ABB RobotStudio station: PaletizadoTPL2.rspag

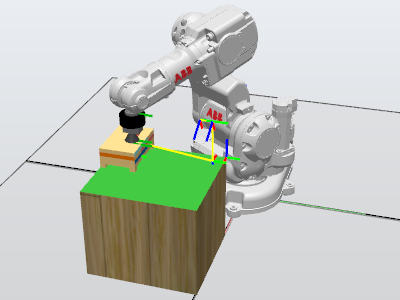
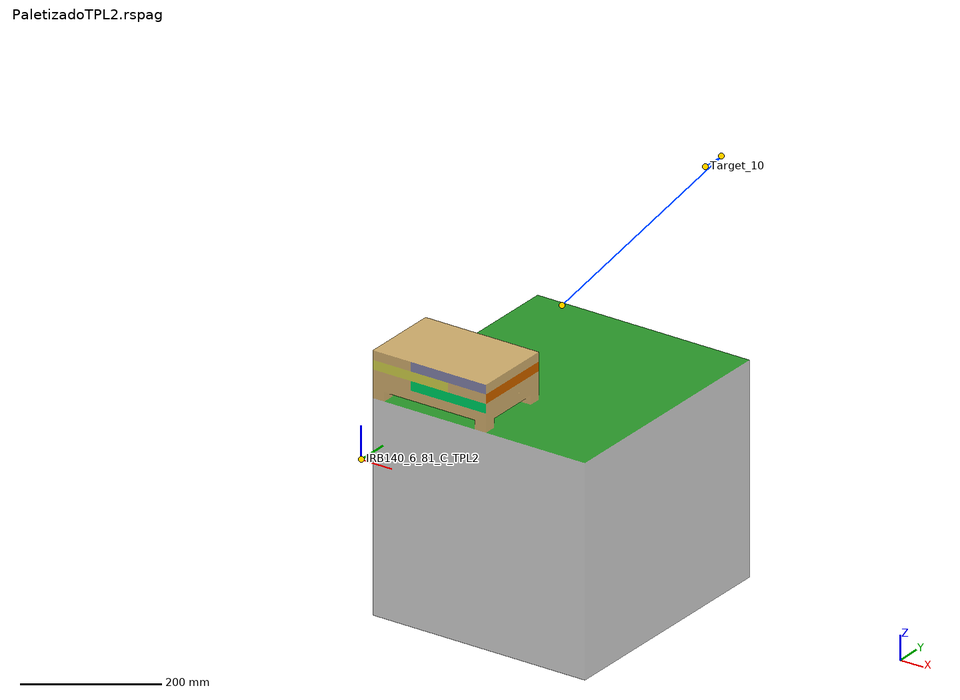
[picture v1: parts stored in the station drawn from their meshes, with robot base, taught points and paths (robot models come from the ABB library and are not in the file)]
--- station ---
Station Paletizado (saved by RobotStudio 25.5.11605.0)
Controller IRB140_6_81_TPL2
  mechanical unit ROB_1: IRB140_6_81_C_TPL2, 6 joints, base frame (0, 0, 0) mm
Layout (positions relative to the parent item):
  - Mesa [part], size 365 x 405 x 340 mm
  - Pallet [part], size 195 x 130 x 30 mm
  - Pieza1 [part] at (65, -275, 60) mm, size 130 x 65 x 15 mm
  - Pieza2 [part] at (795, -395, 45) mm, rotated rx 0 ry 0 rz -180 deg, size 130 x 65 x 15 mm
  - Pieza3 [part] at (305, -700, 30) mm, rotated rx 0 ry 0 rz 90 deg, size 130 x 65 x 15 mm
  - Pieza4 [part] at (730, -395, 0) mm, rotated rx 0 ry 0 rz -180 deg, size 130 x 65 x 15 mm
  - Pieza5 [part] at (0, -275, -15) mm, size 130 x 65 x 15 mm
  - Pieza6 [part] at (490, 30, -30) mm, rotated rx 0 ry 0 rz -90 deg, size 130 x 65 x 15 mm
  - Pieza7 [part] at (65, -275, -60) mm, size 130 x 65 x 15 mm
  - Pieza8 [part] at (795, -395, -75) mm, rotated rx 0 ry 0 rz -180 deg, size 130 x 65 x 15 mm
  - Pieza9 [part] at (305, -700, -90) mm, rotated rx 0 ry 0 rz 90 deg, size 130 x 65 x 15 mm
  - Sopapa [mechanism] at (430, -297.5, 533) mm, rotated rx -180 ry 0 rz 180 deg
      TCP Sopapa at (0, -5, 103) mm
      links: Sopapa
  - IRB140_6_81_C_TPL2 [mechanism, from %ABB.RobotStudio.Models.IRB140%\IRB140_6_81_C_G_03.rslib] at (0, 0, 0) mm; joint values [-0.6052, 0.2446, 0.0306, 0, 1.2955, -0.6052] (rad or m)
Attachment: Sopapa is attached to IRB140_6_81_C_TPL2 / Link6
Attachment: EsquinaPalet is attached to Pallet
EventTableEntry 1212: Group=, Trigger=DO_Sopapa 1213, Actions=[EventTableActionAttach 1214], Comment=, ActivationMode=2, Cyclic=false
EventTableTriggerIO 1213: IOValue=[1], IRC5Controller=? -1, Operator=0, SignalSource=IRB140_6_81_TPL2 1258
EventTableActionAttach 1214: AttachmentParent=Sopapa 1252, AttachmentChild=? -1, MountObject=false, Offset=[X=1, Y=0, Z=0, W=0, X=0, Y=1, Z=0, W=0, X=0, Y=0, Z=1, W=0, X=0, Y=0, Z=0, W=1], FlangeIndext=0, FindNearest=true
EventTableEntry 1219: Group=, Trigger=DO_Sopapa 1220, Actions=[EventTableActionDetach 1221], Comment=, ActivationMode=2, Cyclic=false
EventTableTriggerIO 1220: IOValue=[0], IRC5Controller=? -1, Operator=0, SignalSource=IRB140_6_81_TPL2 1258
EventTableActionDetach 1221: AttachmentParent=Sopapa 1252, AttachmentChild=? -1
EventTableTriggerIO 2360: IOValue=[1], IRC5Controller=? -1, Operator=0, SignalSource=? -1
EventTableTriggerIO 2361: IOValue=[0], IRC5Controller=? -1, Operator=0, SignalSource=? -1
Station signals: DI DO_Sopapa
Targets, tools, work objects and paths stored in the station and not in the controller backup, written as RAPID:
! task T_ROB1
MODULE Module1
  CONST robtarget EsquinaPiezas:=[[405,0,0],[0,0.707106781,0.707106781,0],[0,0,0,0],[9E+09,9E+09,9E+09,9E+09,9E+09,9E+09]];
ENDMODULE


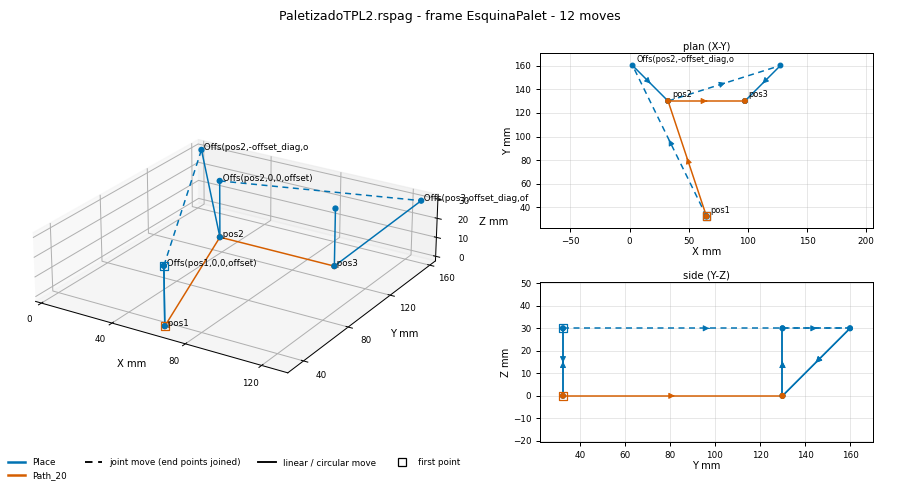
[picture p0: tool path of PaletizadoTPL2.rspag in frame EsquinaPalet, 12 of 19 moves have a stored position in this frame; points joined in program order, loops and branches not executed]
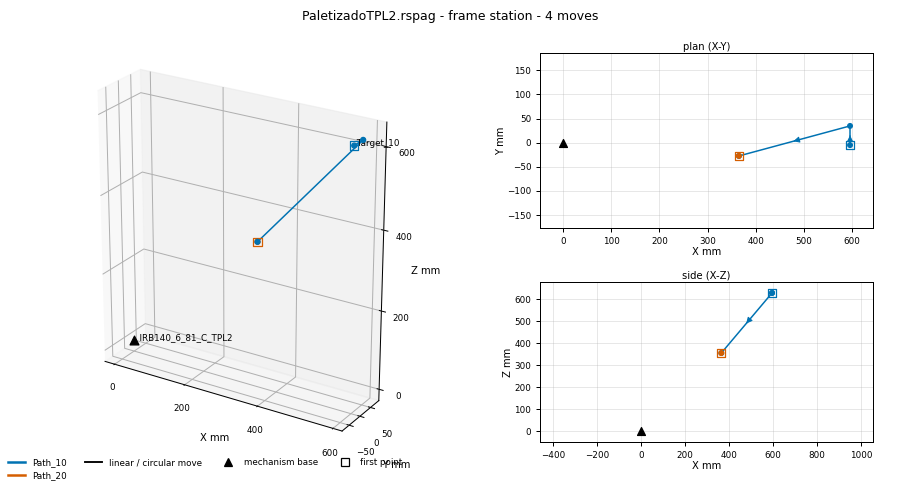
[picture p1: tool path of PaletizadoTPL2.rspag in frame station, 4 of 19 moves have a stored position in this frame; points joined in program order, loops and branches not executed]
--- Backups/IRB140_6_81_TPL2/RAPID/TASK1/PROGMOD/CalibData.mod ---
MODULE CalibData
    PERS wobjdata RefMesa:=[FALSE,TRUE,"",[[300,-400,340],[0,0.707106781,0.707106781,0]],[[0,0,0],[1,0,0,0]]];
    PERS wobjdata EsquinaPalet:=[FALSE,TRUE,"",[[300,-400,370],[0,0.707107,0.707107,0]],[[0,0,-30],[1,0,0,0]]];

ENDMODULE

--- Backups/IRB140_6_81_TPL2/RAPID/TASK1/PROGMOD/Module1.mod ---
MODULE Module1
    PERS tooldata Sopapa:=[TRUE,[[0,-5,103],[1,0,0,0]],[0.5,[0,0,40],[1,0,0,0],0,0,0]];
    CONST robtarget Target_10:=[[595.492267836,-5,628],[0.5,0,0.866025404,0],[0,0,0,0],[9E+09,9E+09,9E+09,9E+09,9E+09,9E+09]];
    CONST robtarget Target_20:=[[595.492192643,34.78927249,628.000011052],[0.500000018,0.000000003,0.866025394,0.000000005],[0,-1,0,0],[9E+09,9E+09,9E+09,9E+09,9E+09,9E+09]];
    CONST robtarget PickPieza:=[[372.5,65,-15],[0.707106781,0,0,-0.707106781],[-1,0,-1,0],[9E+09,9E+09,9E+09,9E+09,9E+09,9E+09]];

    CONST robtarget pos1:=[[65,32.5,0],[0,0,0,1],[-1,0,-2,0],[9E+09,9E+09,9E+09,9E+09,9E+09,9E+09]];
    CONST robtarget pos2:=[[32.5,130,0],[0.707106781,0,0,0.707106781],[-1,0,1,0],[9E+09,9E+09,9E+09,9E+09,9E+09,9E+09]];
    CONST robtarget pos3:=[[97.5,130,0],[0.707106781,0,0,-0.707106781],[-1,0,-1,0],[9E+09,9E+09,9E+09,9E+09,9E+09,9E+09]];


    VAR num CajasEnPalet := 0;
    VAR num PiezasEnPila := 9;


    !Constantes Pieza
    PERS num ancho_pieza := 65;
    PERS num largo_pieza := 130;
    PERS num alto_pieza := 15;

    !Constantes Palet
    PERS num ancho_palet := 130;
    PERS num largo_palet := 195;
    !PERS num alto_palet := 15;

    !Transformacion pinza a perno
    VAR pose sopapa_to_pieza := [[0,0,0], [0,0,0,0]];
    VAR pose transformacion := [[0,0,0], [1,0,0,0]];
    PERS tooldata TCPPieza := [TRUE,[[0,-5,118],[1,0,0,0]],[0.5,[0,0,40],[1,0,0,0],0,0,0]];

    VAR num capa := 0;

    PROC main()
        ConfL\Off;
        ConfJ\Off;

        Init;

        WHILE PiezasEnPila > 0 DO
            Pick;
            Place;
        ENDWHILE

    ENDPROC

    PROC Path_10()
        MoveL Target_10,v1000,z100,Sopapa\WObj:=wobj0;
        MoveL Target_20,v1000,z100,Sopapa\WObj:=wobj0;
        MoveL [[372.5,65,-15],[0.707106781,0,0,-0.707106781],[-1,0,-1,0],[9E+09,9E+09,9E+09,9E+09,9E+09,9E+09]],v1000,z100,Sopapa\WObj:=RefMesa;
    ENDPROC

    PROC Pick()
        VAR num offset := 30;
        MoveJ Offs(PickPieza, 0, 0, -alto_pieza*(PiezasEnPila-1) - offset), v500,z100,Sopapa\WObj:=RefMesa;
        MoveL Offs(PickPieza, 0, 0, -alto_pieza*(PiezasEnPila-1)), v500, fine,Sopapa\WObj:=RefMesa;
        ActivarSopapa;
        WaitTime 1;
        MoveL Offs(PickPieza, 0, 0, -alto_pieza*(PiezasEnPila-1) - offset), v100, fine,Sopapa\WObj:=RefMesa;

    ENDPROC

    PROC Place()
        VAR num offset := -30;
        VAR num offset_diag := 30;

        IF capa MOD 2 = 1 THEN
            transformacion := [[ancho_palet, largo_palet, -alto_pieza*capa],  OrientZYX(180,0,0)];
             !transformacion := [[0, 0, -alto_pieza*capa], [1,0,0,0]];
        ELSE
            transformacion := [[0, 0, -alto_pieza*capa], [1,0,0,0]];
        ENDIF

        EsquinaPalet.oframe := transformacion;

        TEST CajasEnPalet MOD 3

            CASE 0:
                MoveJ Offs(pos1, 0, 0, offset), v500,z100,TCPPieza\WObj:=EsquinaPalet;
                MoveL pos1, v100, fine,TCPPieza\WObj:=EsquinaPalet;
                DesactivarSopapa;
                WaitTime 1;
                CajasEnPalet := CajasEnPalet + 1;
                PiezasEnPila := PiezasEnPila - 1;
                MoveL Offs(pos1, 0, 0, offset), v100, z100,Sopapa\WObj:=EsquinaPalet;

            CASE 1:
                MoveJ Offs(pos2, -offset_diag, offset_diag, offset), v500,fine,TCPPieza\WObj:=EsquinaPalet;
                MoveL pos2, v100, fine,TCPPieza\WObj:=EsquinaPalet;
                DesactivarSopapa;
                WaitTime 1;
                CajasEnPalet := CajasEnPalet + 1;
                PiezasEnPila := PiezasEnPila - 1;
                MoveL Offs(pos2, 0, 0, offset), v100, z100,Sopapa\WObj:=EsquinaPalet;

            CASE 2:
                MoveJ Offs(pos3, offset_diag, offset_diag, offset), v500,fine,TCPPieza\WObj:=EsquinaPalet;
                MoveL pos3, v100, fine,TCPPieza\WObj:=EsquinaPalet;
                DesactivarSopapa;
                WaitTime 1;
                CajasEnPalet := CajasEnPalet + 1;
                PiezasEnPila := PiezasEnPila - 1;
                MoveL Offs(pos3, 0, 0, offset), v100, z100,Sopapa\WObj:=EsquinaPalet;
                capa := capa + 1;

        ENDTEST

    ENDPROC

    PROC Init()

        CajasEnPalet := 0;
        PiezasEnPila := 9;

        DesactivarSopapa;
        !sopapa_to_pieza := [[-largo_pieza/2,ancho_pieza/2,0],  OrientZYX(0,0,0)];
        sopapa_to_pieza := [[0,0, alto_pieza],  OrientZYX(0,0,0)];
        TCPPieza.tframe := PoseMult(Sopapa.tframe, sopapa_to_pieza);


    ENDPROC

    PROC ActivarSopapa()
        SetDO DO_Sopapa,1;
    ENDPROC

    PROC DesactivarSopapa()
        SetDO DO_Sopapa,0;
    ENDPROC

    PROC Path_20()
        MoveL [[372.5,65,-15],[0.707106781,0,0,-0.707106781],[-1,0,-1,0],[9E+09,9E+09,9E+09,9E+09,9E+09,9E+09]],v1000,z100,Sopapa\WObj:=RefMesa;
        MoveL pos1,v1000,z100,Sopapa\WObj:=EsquinaPalet;
        MoveL pos2,v1000,z100,Sopapa\WObj:=EsquinaPalet;
        MoveL pos3,v1000,z100,Sopapa\WObj:=EsquinaPalet;
    ENDPROC




ENDMODULE

--- Backups/IRB140_6_81_TPL2/RAPID/TASK1/SYSMOD/LINKEDM.sys ---
%%%
  VERSION:1
  LANGUAGE:ENGLISH
%%%

MODULE LINKEDM (SYSMODULE)

! FOLLOWER
!     Name of electronically linked follower axis used by operator at teach pendent.
      PERS string l_f_axis_name{5}       :=  ["",  "", "", "", ""];

!     Name of the mechanical unit for follower axis.
      PERS string l_f_mecunt_n{5}  :=  ["", "", "", "", ""];

!     Linked follower axis number in the mechanical unit (first axis in mech. unit is number 1).
      PERS num l_f_axis_no{5}      :=  [0,          0,   0,  0,  0];

! MASTER
!     Name of the mechanical unit for linked master axis.
      PERS string l_m_mecunt_n{5} :=  ["", "", "", "", ""];

!     Linked master axis number in the mechanical unit (first axis in mech. unit is number 1).
!     See axis number table in documentation for different master mechanical units.
      PERS num l_m_axis_no{5}     :=  [0,  0,  0,  0,  0];

! POSITION OFFSET
!     The increase of the allowed offset position between the master and follower
!     positions, used when starting AUTO mode. As soon as the offset is decreased
!     the old configurated parameter is used.
!     Example: 3 => the configurated value of allowed offset is increased 3 times.
      PERS num offset_ratio{5}       :=  [10,  10,   10,  10,  10];

! SPEED RATIO
!     Speed_ratio used in AUTO and JOG modes [ very_slow   slow    normal    fast]
!     Value 1 = max allowed manual speed.
      CONST num speed_ratio {20}      := [0.01, 0.01, 0.01, 0.01, 0.01,
                                          0.05, 0.05, 0.05, 0.05, 0.05,
                                          0.20, 0.20, 0.20, 0.20, 0.20,
                                          1.00, 1.00, 1.00, 1.00, 1.00];

! STEP SIZE
!     Displacement position used in JOG mode for each activation of positive or
!     negative movement.                  [very_short    short   normal   long]
!     Unit degees or meter.
      CONST num displacement {20}     := [0.001, 0.001, 0.001, 0.001, 0.001,
                                          0.005, 0.005, 0.005, 0.005, 0.005,
                                          0.020, 0.020, 0.020, 0.020, 0.020,
                                          0.100, 0.100, 0.100, 0.100, 0.100];


!-------------------------------------------------------------
 PROC Linked_m ()
      Linked_m_exe ;
 ENDPROC
ENDMODULE

--- Backups/IRB140_6_81_TPL2/SYSPAR/EIO.cfg ---
EIO:CFG_1.0:6:1::
#
EIO_SIGNAL:

      -Name "DO_Sopapa" -SignalType "DO"
